Universal Robots PolyScope program: pickPlace_v1_grp6.urp

Program pickPlace_v1_grp6 (installation=default directory=/programs createdIn=5.17.2 lastSavedIn=5.17.2 robotSerialNumber=20195300624)
Calibrated DH parameters: a=[-0.000114, -0.243449, -0.156545, 0.000118, -0.000132, 0]; d=[0.151995, 1.791478, 30.860003, -32.520701, 0.085404, 0.092246]; alpha=[1.571702, -0.004219, 0.004452, 1.571799, -1.572316, 0]; deltaTheta=[0, -0.031039, 0.779457, -0.748425, -0.000001, 0]
InitVariablesNode variables(variable(name=PLOC_Ref, expression=[0.000000,-1.570800,-1.570800,-1.745330,1.570800,1.570800]), variable(name=PLOC_clear, expression=p[0,0,0,0,0,0]), variable(name=PLOC_pick, expression=p[0,0,0,0,0,0]), variable(name=PLOC_prepick, expression=[0,0,0,0,0,0]), variable(name=PLOC_total, expression=0), variable(name=PLOC_total_1, expression=0))
Robot Program (runOnlyOnce=false)
  URCap PLOC2D (PART LOCALIZATION WITH SICK PLOC2D, SICK AG - Developed by Nimalendiran Kailasanathan) dataModel(Z_OFFSET=0.0, IS_PICK_ALL_PARTS_SELECTED=1, LOCALIZATION_TIMEOUT=1, IS_ABOVE_BIN_SET_KEY=true, IP_ADDRESS_LIST_OF=[10.0.120.31], SELECTED_JOBS=2 , SELECTED_IP_ADDRESS=10.0.120.31, SELECTED_ALIGNMENT_NAME=ploc_align_grp6, Variable(key=PLOC_REF_POSE_KEY, variable(name=PLOC_Ref, initializeExpression=[0.000000,-1.570800,-1.570800,-1.745330,1.570800,1.570800])), Variable(key=PLOC_PRE_PICK_POSE, variable(name=PLOC_prepick, initializeExpression=[0,0,0,0,0,0])), Variable(key=PLOC_PICK_POSE, variable(name=PLOC_pick, initializeExpression=p[0,0,0,0,0,0])), Variable(key=PLOC_CLEAR_POSE_KEY, variable(name=PLOC_clear, initializeExpression=p[0,0,0,0,0,0])), Variable(key=TOTAL_VAR, variable(name=PLOC_total, initializeExpression=0)), Variable(key=NUMBER_OF_MATCHES_VAR, variable(name=PLOC_total_1, initializeExpression=0)), TCP(key=selected-tcp name=GripperClosed), JointPositions(key=JOINT_REF_ANGLES, JointPosition(key=[1], Angle(key=pos value=0.21141 unit=RAD)), JointPosition(key=[2], Angle(key=pos value=-0.9031 unit=RAD)), JointPosition(key=[3], Angle(key=pos value=1.41767 unit=RAD)), JointPosition(key=[4], Angle(key=pos value=-2.9779 unit=RAD)), JointPosition(key=[5], Angle(key=pos value=3.8959 unit=RAD)), JointPosition(key=[6], Angle(key=pos value=0.58522 unit=RAD))), Pose(key=SELECTED_ALIGNMENT_POSE, Position(key=posePosition, Length(key=X value=-0.45985 unit=M), Length(key=Y value=-0.07307 unit=M), Length(key=Z value=0.09953 unit=M)), Rotation(key=poseRotation, Angle(key=RX value=2.89649 unit=RAD), Angle(key=RY value=-1.19701 unit=RAD), Angle(key=RZ value=-0.01175 unit=RAD))))
    Folder Pick and Place
      Folder Start
        'Set start position and open gripper'
        MoveJ speed 60 deg/s, acceleration 80 deg/s^2 (useActiveTCP=false) tcp=GripperClosed; feature=Base
          Waypoint Start: motionParameters(blendRadius=0); TCP in base x=-365.872 y=51.788 z=144.759 mm, rx=0.0967 ry=-3.0002 rz=-0.1965 rad; joints [-26.724, -103.085, 106.736, -134.954, 265.61, 4.947] deg; TCP offset x=-0.756 y=92.532 z=208.204 mm, rx=-0.3257 ry=-0.5801 rz=-2.1551 rad
        URCap RG Grip (OnRobot, OnRobot A/S) dataModel(rg-target-force=8.0, payload-weight=0.0, workpiece-lost=false, rg-target-width=0.036000000000000004, Variable(key=on_return, variable(name=on_return)))
      current_pose := get_actual_tcp_pose()
      pick_pose := p[PLOC_pick[0],PLOC_pick[1],PLOC_pick[2],current_pose[3],current_pose[4],current_pose[5]]
      prePick_pose := p[pick_pose[0],pick_pose[1],pick_pose[2]+0.0500,pick_pose[3],pick_pose[4],pick_pose[5]]
      Popup Message (haltProgram=false inputType=Variable) variable=prePick_pose
      Folder Approach
        MoveJ speed 60 deg/s, acceleration 80 deg/s^2 (useActiveTCP=false) tcp=GripperClosed; feature=Base
          Waypoint Variable (Variable): motionParameters(blendRadius=0.01); variable=prePick_pose
      Popup Message (haltProgram=false inputType=Variable) variable=pick_pose
      Folder Pick
        MoveL speed 250 mm/s, acceleration 1200 mm/s^2 (useActiveTCP=false) tcp=GripperClosed; feature=Base
          Waypoint Variable (Variable): variable=pick_pose
        URCap RG Grip (OnRobot, OnRobot A/S) dataModel(rg-target-force=8.0, payload-weight=0.0, workpiece-lost=false, rg-target-width=0.0127, Variable(key=on_return, variable=on_return))
      Folder Clear
        'Close gripper'
        MoveL speed 250 mm/s, acceleration 1200 mm/s^2 (useActiveTCP=false) tcp=GripperClosed; feature=Base
          Waypoint Variable (Variable): motionParameters(blendRadius=0.01); variable=prePick_pose
      Popup Message (haltProgram=false inputType=Variable) variable=prePick_pose
      Folder Place
        'Set drop position and open gripper'
        SuppressedNode
          MoveJ speed 60 deg/s, acceleration 80 deg/s^2 (useActiveTCP=false) tcp=GripperClosed; feature=Base
            Waypoint Place: motionParameters(blendRadius=0); TCP in base x=-262.248 y=-239.165 z=198.59 mm, rx=1.6242 ry=-2.5509 rz=0.0228 rad; joints [12.158, -106.29, 90.65, -110.461, 282.127, -10.952] deg
        SuppressedNode
          MoveJ speed 60 deg/s, acceleration 80 deg/s^2 (useActiveTCP=true) feature=Base
            Waypoint Waypoint_2: TCP in base x=-323.834 y=-253.208 z=163.159 mm, rx=1.3176 ry=-2.6657 rz=-0.1012 rad; joints [21.198, -92.423, 92.377, -130.816, 266, 4.013] deg
        SuppressedNode
          MoveJ speed 60 deg/s, acceleration 80 deg/s^2 (useActiveTCP=true) feature=Base
            Waypoint Waypoint_1: TCP in base x=-336.523 y=-254.12 z=93.116 mm, rx=1.3176 ry=-2.6657 rz=-0.1012 rad; joints [20.456, -87.145, 106.283, -150.041, 266.383, 3.432] deg
        URCap RG Grip (OnRobot, OnRobot A/S) dataModel(rg-target-force=8.0, payload-weight=0.0, workpiece-lost=false, rg-target-width=0.036000000000000004, Variable(key=on_return, variable=on_return))
  SuppressedNode
    MoveJ speed 60 deg/s, acceleration 80 deg/s^2 (useActiveTCP=true) feature=Base
      Waypoint Waypoint_3: TCP in base x=-280.783 y=-121.18 z=407.203 mm, rx=-0.6447 ry=-0.6232 rz=1.4456 rad; joints [-2.632, -104.605, 96.863, -125.662, 270.543, -0.096] deg; TCP offset x=0 y=0 z=0 mm, rx=1.5708 ry=0 rz=0 rad
      Wait Sleep waitTime=1
      Waypoint Waypoint_6: TCP in base x=-275.071 y=102.503 z=235.011 mm, rx=-1.0353 ry=-2.575 rz=0.8337 rad; joints [-32.174, -84.485, 106.989, -97.093, 217.926, -69.873] deg
      Wait Sleep waitTime=2
      Waypoint Waypoint_7: TCP in base x=-292.982 y=108.647 z=184.415 mm, rx=-0.9436 ry=-2.3391 rz=0.3899 rad; joints [-29.841, -72.73, 112.336, -115.307, 208.528, -46.542] deg
      Wait Sleep waitTime=2
      Waypoint Waypoint_4: TCP in base x=-192.949 y=44.324 z=168.925 mm, rx=0.7131 ry=1.6105 rz=-0.5324 rad; joints [-26.025, -72.75, 112.319, -31.073, 199.862, -72.807] deg
      Wait Sleep waitTime=2
      Set NoAction
      Waypoint Waypoint_5: TCP in base x=-49.853 y=-250.493 z=441.7 mm, rx=-0.2982 ry=-0.7807 rz=2.2996 rad; joints [47.11, -117.219, 100.254, -125.66, 270.545, -0.098] deg
